// TIA Portal V19 export
TYPE "LUC_typeModeState"
TITLE = LUC_typeModeState
// Duration of stay in one mode and state
// stored: Access Published
   STRUCT
      mode { ExternalWritable := 'False'} : DInt;   // OMAC identifier of mode
      state { ExternalWritable := 'False'} : DInt;   // OMAC identifier of state
      duration { ExternalWritable := 'False'} : LReal;   // Time stayed in that status
   END_STRUCT;
END_TYPE
